// TIA Portal V18 export
DATA_BLOCK "L1_VitaPunzoni"   // DB40
{ S7_Optimized_Access := 'TRUE' }
VERSION : 0.1
// stored: AutoNumber false, DBAccessibleFromOPCUA true, DBAccessibleFromWebserver true, IsOnlyStoredInLoadMemory false, IsRetainMemResEnabled false, IsWriteProtectedInAS false, MemoryReserve 100
   VAR RETAIN
      Punzonatura : Struct   // vita punzoni banco di punzonatura
         Stampo : Array[1..32] of DInt;
         Cassetto : Array[1..64] of DInt;
      END_STRUCT;
      Plotter : Struct   // vita punzoni cassetti del plotter
         Cassetto : Array[1..32] of DInt;
      END_STRUCT;
      Taglio : Struct   // vita punzoni postpunzonatura o taglio al volo
         Stampo : Array[1..16] of DInt;   // vita punzoni taglio
         Cassetto : Array[1..16] of DInt;
      END_STRUCT;
      Generico : Struct   // vita punzoni stampi vari
         Stampo : Array[1..16] of DInt;
         Cassetto : Array[1..16] of DInt;
      END_STRUCT;
   END_VAR
BEGIN
END_DATA_BLOCK
